SUBAPPLICATION QualityCamera (* Subapplication Type *)
  (* Standard: 61499-2 *)
  (* Version 1.0, 2025-03-21, AK123700 *)
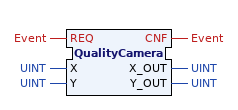
  EVENT_INPUT
    REQ; (* Normal Execution Request *)
  END_EVENT
  EVENT_OUTPUT
    CNF; (* Execution Confirmation *)
  END_EVENT
  VAR_INPUT
    X : UINT; (* Input event qualifier *)
    Y : UINT;
  END_VAR
  VAR_OUTPUT
    X_OUT : UINT; (* Output event qualifier *)
    Y_OUT : UINT;
  END_VAR
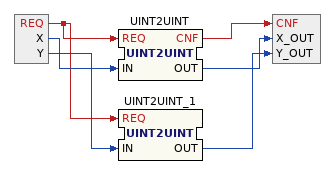
  FBS
    UINT2UINT : UINT2UINT;
    UINT2UINT_1 : UINT2UINT;
  END_FBS
  EVENT_CONNECTIONS
    REQ TO UINT2UINT.REQ;
    REQ TO UINT2UINT_1.REQ;
    UINT2UINT.CNF TO CNF;
  END_CONNECTIONS
  DATA_CONNECTIONS
    X TO UINT2UINT.IN;
    Y TO UINT2UINT_1.IN;
    UINT2UINT_1.OUT TO Y_OUT;
    UINT2UINT.OUT TO X_OUT;
  END_CONNECTIONS
END_SUBAPPLICATION
